FUNCTION_BLOCK FB_ClearConveyer
VAR_INPUT
	Execute : BOOL;
END_VAR
VAR_OUTPUT
END_VAR
VAR
	

	stopTimer				: TON;	
	fbStop					: MC_Stop;
	bVelocityExecute		: BOOL;
	conveyerVelocity		: LREAL := 800;
	nState					: INT := -2;
	Done					: BOOL;
	bStopExecute			: BOOL;
	bTimerStart				: BOOL;
	fbMoveVelocity			: MC_MoveVelocity;
	direction				: TC2_MC2.MC_Direction;
END_VAR

fbMoveVelocity(
	Axis:= GVL_Conveyer.ConveyerAxis, 
	Execute:= bVelocityExecute, 
	Velocity:= conveyerVelocity, 
	Direction := direction
	 );

stopTimer(
	IN := bTimerStart,
	PT := T#1S
	);

fbStop(
	Axis:= GVL_Conveyer.ConveyerAxis, 
	Execute:= bStopExecute,
	);
		
bVelocityExecute := FALSE;
bStopExecute 	 := FALSE;


IF Execute THEN
	
	CASE nState OF
		
		-2:
			bStopExecute := TRUE;
			nState := -1;
			
		-1:
			IF fbStop.Done THEN
				nState := 0;
			END_IF
		

		0:
			direction := MC_Negative_Direction;
			bVelocityExecute := TRUE;
			nState := 1;
			
		1:
			bTimerStart := TRUE;
			IF stopTimer.Q THEN
				bTimerStart := FALSE;
				bStopExecute := TRUE;
				nState := 2;
			END_IF
		2:
			IF fbStop.Done THEN
				bVelocityExecute := TRUE;
				direction := MC_Positive_Direction;
				nState := 3;
			END_IF
			
			
			
		3:
			bTimerStart := TRUE;
			IF stopTimer.Q THEN
				bTimerStart := FALSE;
				nState := 4;
			END_IF
		
		4:
			GVL.bPuckMissed := FALSE;
			GVL.bClearPuck := FALSE;
			Done := TRUE;
	
	
	END_CASE

ELSE
	Done := FALSE;
	nState := -2;
END_IF

END_FUNCTION_BLOCK

(* stored: Version 1.1.0.1, ProductVersion 3.1.4024.11
   POU FB_ClearConveyer: Id {161a3070-fb25-49b3-89f5-5450182cb1ff}, SpecialFunc None *)
